// TwinCAT 3 PLC project BaseFBs
// Title: BaseFBs
// Company: Personal
// ProjectVersion: 1.0.0.3
// ProgramVersion: 3.1.4026.14
// libraries:
//   Tc2_Standard, * (Beckhoff Automation GmbH)
//   Tc2_System, * (Beckhoff Automation GmbH)
// project tree:
//   FBs/ FB_Base.TcPOU, FB_EquipmentBase.TcPOU, FB_Alarm.TcPOU, FB_SupervisorBase.TcPOU, ITF_Base.TcIO, ITF_EquipmentBase.TcIO, ITF_SupervisorBase.TcIO, Param_SupervisorBase.TcGVL
//   FBs/Structure/ ST_BaseDefinition.TcDUT, ST_EquipmentAlarm.TcDUT, ST_EquipmentAlarmListDetails.TcDUT
//   / PlcTask.TcTTO
//   POUs/ MAIN.TcPOU
//   TestFBs/TestBase/ FB_TestBase.TcPOU
//   TestFBs/TestEquipmentBase/ E_TestEquipmentAlarmList.TcDUT, FB_TestEquipmentBase.TcPOU
// real-time tasks:
//   TASK PlcTask: cycle T#10ms, priority 20, ADS port 350

CONFIGURATION BaseFBs
    RESOURCE PLC ON TwinCAT3
        TASK PlcTask(INTERVAL := T#10ms, PRIORITY := 20);
        PROGRAM MAIN WITH PlcTask : MAIN;
    END_RESOURCE
END_CONFIGURATION

// ---- FBs/Structure/ST_BaseDefinition.TcDUT
TYPE ST_BaseDefinition :
STRUCT
	Name		: STRING(40);
	Station		: string(40);
END_STRUCT
END_TYPE

// ---- FBs/Structure/ST_EquipmentAlarm.TcDUT
TYPE ST_EquipmentAlarm :
STRUCT
	Active			: BOOL;
	Message			: T_MaxString;
	Severity		: TcEventSeverity;
END_STRUCT
END_TYPE

// ---- FBs/Structure/ST_EquipmentAlarmListDetails.TcDUT
TYPE ST_EquipmentAlarmListDetails :
STRUCT
	FirstAlarm		: POINTER TO ST_EquipmentAlarm;
	AlarmListSize	: DINT; 
END_STRUCT
END_TYPE

// ---- TestFBs/TestEquipmentBase/E_TestEquipmentAlarmList.TcDUT
{attribute 'qualified_only'}
{attribute 'strict'}
{attribute 'to_string'}
TYPE E_TestEquipmentAlarmList :
(
	VerboseAlarm,
	InfoAlarm,
	WarningAlarm,
	ErrorAlarm,
	CriticalAlarm
);
END_TYPE

// ---- FBs/Param_SupervisorBase.TcGVL
{attribute 'qualified_only'}
VAR_GLOBAL CONSTANT
	AlarmListSize	: DINT := 50;
END_VAR

// ---- FBs/ITF_Base.TcIO
INTERFACE ITF_Base

PROPERTY Definition : REFERENCE TO ST_BaseDefinition
GET
END_GET
END_PROPERTY

PROPERTY EnableManualControl : Bool
SET
END_SET
END_PROPERTY

END_INTERFACE

// ---- FBs/ITF_EquipmentBase.TcIO
  INTERFACE ITF_EquipmentBase EXTENDS ITF_Base

PROPERTY AlarmListDetails : Reference to ST_EquipmentAlarmListDetails
GET
END_GET
END_PROPERTY

PROPERTY MainAlarm : Reference to ST_EquipmentAlarm
GET
END_GET
END_PROPERTY

METHOD Reset
END_METHOD

END_INTERFACE

// ---- FBs/ITF_SupervisorBase.TcIO
INTERFACE ITF_SupervisorBase

METHOD CheckAlarmCondition
VAR_INPUT
	AlarmToRaise		: ST_EquipmentAlarm;
	ConcatenateMessage	: T_MaxString;
END_VAR
END_METHOD

METHOD CheckAlarmConditionCustom
VAR_INPUT
	Active	: BOOL;
	Message	: T_MaxString;
	Severity	: TcEventSeverity;
END_VAR
END_METHOD

METHOD CompileAlarmList
VAR_INPUT
	AlarmListDetails		: ST_EquipmentAlarmListDetails;
END_VAR
END_METHOD

END_INTERFACE

// ---- POUs/MAIN.TcPOU
PROGRAM MAIN
VAR
	fbTestBase : FB_TestBase;
	fbTestEquipmentBase	: FB_TestEquipmentBase;
	fbTestEquipmentBase2	: FB_TestEquipmentBase;
	
	AnotherTestAlarmList	: ARRAY[E_TestEquipmentAlarmList.VerboseAlarm..E_TestEquipmentAlarmList.CriticalAlarm] OF ST_EquipmentAlarm;
	
	Reset	: BOOL;
	
	fbSupervistorBase : FB_SupervisorBase;
	
END_VAR

VAR PERSISTENT
	TestManualControl	: ARRAY[1..3] OF BOOL;
	TestName			: ARRAY[1..3] OF STRING(40);
	TestStation			: ARRAY[1..3] OF STRING(40);	
	

END_VAR

fbTestBase.Definition.Name := TestName[1];
fbTestBase.Definition.Station := TestStation[1];
fbTestBase.EnableManualControl := TestManualControl[1];

fbTestBase();

fbTestEquipmentBase.Definition.Name := TestName[2];
fbTestEquipmentBase.Definition.Station := TestStation[2];
fbTestEquipmentBase.EnableManualControl := TestManualControl[2];

fbTestEquipmentBase();

fbTestEquipmentBase2.Definition.Name := TestName[3];
fbTestEquipmentBase2.Definition.Station := TestStation[3];
fbTestEquipmentBase2.EnableManualControl := TestManualControl[3];

fbTestEquipmentBase2();

IF Reset THEN
	fbTestEquipmentBase.Reset();	
	fbTestEquipmentBase2.Reset();
	Reset := FALSE;
END_IF

fbSupervistorBase();

fbSupervistorBase.CompileAlarmList(AlarmListDetails := fbTestEquipmentBase.AlarmListDetails);
fbSupervistorBase.CompileAlarmList(AlarmListDetails := fbTestEquipmentBase2.AlarmListDetails);

END_PROGRAM

// ---- TestFBs/TestBase/FB_TestBase.TcPOU
FUNCTION_BLOCK FB_TestBase EXTENDS FB_Base

VAR
END_VAR

END_FUNCTION_BLOCK

// ---- FBs/FB_Base.TcPOU
FUNCTION_BLOCK ABSTRACT FB_Base IMPLEMENTS ITF_Base
VAR
	_Definition				: ST_BaseDefinition;
	_EnableManualControl	: BOOL;
END_VAR

PROPERTY Definition : REFERENCE TO ST_BaseDefinition
GET
Definition REF= _Definition;
END_GET
END_PROPERTY

PROPERTY EnableManualControl : BOOL
SET
_EnableManualControl := EnableManualControl;
END_SET
END_PROPERTY

END_FUNCTION_BLOCK

// ---- TestFBs/TestEquipmentBase/FB_TestEquipmentBase.TcPOU
FUNCTION_BLOCK FB_TestEquipmentBase EXTENDS FB_EquipmentBase
VAR
	TestAlarmList	: ARRAY[E_TestEquipmentAlarmList.VerboseAlarm..E_TestEquipmentAlarmList.CriticalAlarm] OF ST_EquipmentAlarm;
	
	AlarmType		: E_TestEquipmentAlarmList;
	RaiseAlarmFlag	: BOOL;
END_VAR


SUPER^();
fbAlarm(AlarmList := TestAlarmList);

IF RaiseAlarmFlag THEN
	
	CASE AlarmType OF
		E_TestEquipmentAlarmList.VerboseAlarm:
			_RaiseAlarm(AlarmToRaise := TestAlarmList[E_TestEquipmentAlarmList.VerboseAlarm], ConcatenateMessage := '');
		
		E_TestEquipmentAlarmList.InfoAlarm:
			_RaiseAlarm(AlarmToRaise := TestAlarmList[E_TestEquipmentAlarmList.InfoAlarm], ConcatenateMessage := '');
		
		E_TestEquipmentAlarmList.WarningAlarm:
			_RaiseAlarm(AlarmToRaise := TestAlarmList[E_TestEquipmentAlarmList.WarningAlarm], ConcatenateMessage := '');
		
		E_TestEquipmentAlarmList.ErrorAlarm:
			_RaiseAlarm(AlarmToRaise := TestAlarmList[E_TestEquipmentAlarmList.ErrorAlarm], ConcatenateMessage := '');
		
		E_TestEquipmentAlarmList.CriticalAlarm:
			_RaiseAlarm(AlarmToRaise := TestAlarmList[E_TestEquipmentAlarmList.CriticalAlarm], ConcatenateMessage := '');
		
	END_CASE

	RaiseAlarmFlag := FALSE;
END_IF

{warning 'Add method implementation '}
METHOD PROTECTED _GenerateAlarmList
TestAlarmList[E_TestEquipmentAlarmList.VerboseAlarm].Message 		:= 'Verbose Alarm';
TestAlarmList[E_TestEquipmentAlarmList.VerboseAlarm].Severity 		:= TcEventSeverity.Verbose;

TestAlarmList[E_TestEquipmentAlarmList.InfoAlarm].Message 			:= 'Info Alarm';
TestAlarmList[E_TestEquipmentAlarmList.InfoAlarm].Severity 			:= TcEventSeverity.Info;

TestAlarmList[E_TestEquipmentAlarmList.WarningAlarm].Message 		:= 'Warning Alarm';
TestAlarmList[E_TestEquipmentAlarmList.WarningAlarm].Severity 		:= TcEventSeverity.Warning;

TestAlarmList[E_TestEquipmentAlarmList.ErrorAlarm].Message 			:= 'Error Alarm';
TestAlarmList[E_TestEquipmentAlarmList.ErrorAlarm].Severity 		:= TcEventSeverity.Error;

TestAlarmList[E_TestEquipmentAlarmList.CriticalAlarm].Message 		:= 'Critical Alarm';
TestAlarmList[E_TestEquipmentAlarmList.CriticalAlarm].Severity 		:= TcEventSeverity.Critical;
END_METHOD

END_FUNCTION_BLOCK

// ---- FBs/FB_EquipmentBase.TcPOU
FUNCTION_BLOCK ABSTRACT FB_EquipmentBase EXTENDS FB_Base IMPLEMENTS ITF_EquipmentBase

VAR
	fbAlarm		: FB_Alarm;
	_MainAlarm	: ST_EquipmentAlarm;
	_AlarmListDetails	: ST_EquipmentAlarmListDetails;
	AlarmListUpperBound		: DINT;
	AlarmListLowerBound		: DINT;
	EmptyAlarmList			: BOOL;
	
	EquipmentBaseFirstScan	: BOOL := TRUE;
	
END_VAR

fbAlarm.Definition.Name := _Definition.Name;

_AlarmListDetails := fbAlarm.AlarmListDetails;

IF EquipmentBaseFirstScan THEN
	_GenerateAlarmList();
END_IF

EquipmentBaseFirstScan := FALSE;

METHOD PROTECTED _GenerateAlarmList
END_METHOD

METHOD PROTECTED _RaiseAlarm
VAR_INPUT
	AlarmToRaise	: REFERENCE TO ST_EquipmentAlarm;
	ConcatenateMessage	: T_MaxString;
END_VAR
AlarmToRaise.Active := TRUE;

IF (NOT _MainAlarm.Active) OR (AlarmToRaise.Severity > _MainAlarm.Severity) THEN
	_MainAlarm := AlarmToRaise;
	
	IF ConcatenateMessage <> '' THEN
		_MainAlarm.Message := CONCAT(STR1 := _MainAlarm.Message, STR2 := ConcatenateMessage);
	END_IF
	
END_IF
END_METHOD

{warning 'Add property implementation'}
PROPERTY AlarmListDetails : REFERENCE TO ST_EquipmentAlarmListDetails
GET
 AlarmListDetails REF= _AlarmListDetails;
END_GET
END_PROPERTY

{warning 'Add property implementation'}
PROPERTY MainAlarm : REFERENCE TO ST_EquipmentAlarm
GET
MainAlarm REF= _MainAlarm;
END_GET
END_PROPERTY

{warning 'Add method implementation '}
METHOD Reset
VAR
	ErrorIndex	: DINT;
END_VAR
_MainAlarm.Active := FALSE;
_MainAlarm.Severity := TcEventSeverity.Verbose;
_MainAlarm.Message := '';

fbAlarm.Reset();
END_METHOD

END_FUNCTION_BLOCK

// ---- FBs/FB_Alarm.TcPOU
FUNCTION_BLOCK  FB_Alarm EXTENDS FB_Base IMPLEMENTS ITF_Base
VAR_IN_OUT
	AlarmList	: ARRAY[*] OF ST_EquipmentAlarm;
END_VAR
VAR
	_AlarmListDetails	: ST_EquipmentAlarmListDetails;
	AlarmListUpperBound		: DINT;
	AlarmListLowerBound		: DINT;
	EmptyAlarmList			: BOOL;
	
	AlarmIndex				: DINT;
	DefinitionNameScanned	: BOOL := FALSE;
	
	FirstScan	: BOOL := TRUE;
END_VAR

_AlarmListHandling();

IF _Definition.Name <> '' AND not DefinitionNameScanned THEN
	
	FOR AlarmIndex := AlarmListLowerBound TO AlarmListUpperBound BY 1 DO
		AlarmList[AlarmIndex].Message := CONCAT(STR1 := ': ', STR2 := AlarmList[AlarmIndex].Message);
		AlarmList[AlarmIndex].Message := CONCAT(STR1 := _Definition.Name, STR2 := AlarmList[AlarmIndex].Message);
	END_FOR
	
	DefinitionNameScanned := TRUE;
END_IF

FirstScan := FALSE;

METHOD Private _AlarmListHandling

EmptyAlarmList := FALSE;
IF (SIZEOF(AlarmList) = 0) OR (AlarmList = 0) THEN
	EmptyAlarmList := TRUE;
	RETURN;
END_IF
	
IF FirstScan THEN	
	AlarmListLowerBound := LOWER_BOUND(AlarmList,1);
	AlarmListUpperBound := UPPER_BOUND(AlarmList,1);
	
	_AlarmListDetails.AlarmListSize := AlarmListUpperBound - AlarmListLowerBound + 1;
	_AlarmListDetails.FirstAlarm := ADR(AlarmList[AlarmListLowerBound]);
	
END_IF
END_METHOD

{warning 'Add property implementation'}
PROPERTY AlarmListDetails : REFERENCE TO ST_EquipmentAlarmListDetails
GET
 AlarmListDetails REF= _AlarmListDetails;
END_GET
END_PROPERTY

{warning 'Add method implementation '}
METHOD Reset
VAR
	ErrorIndex	: DINT;
END_VAR
IF EmptyAlarmList THEN
	RETURN;
END_IF

FOR ErrorIndex := AlarmListLowerBound TO AlarmListUpperBound BY 1 DO
	AlarmList[ErrorIndex].Active := FALSE;
END_FOR
END_METHOD

END_FUNCTION_BLOCK

// ---- FBs/FB_SupervisorBase.TcPOU
FUNCTION_BLOCK FB_SupervisorBase EXTENDS FB_EquipmentBase IMPLEMENTS ITF_SupervisorBase
VAR
	CompiledAlarm, CompiledAlarm_Intermediate		: ARRAY[0..Param_SupervisorBase.AlarmListSize] OF ST_EquipmentAlarm;	
	EmptyAlarm						: ST_EquipmentAlarm;	
	AlarmListIndex					: DINT;
	index							: DINT;
END_VAR

SUPER^();

_ResetAlarmList();

METHOD PRIVATE _ResetAlarmList
VAR_INPUT
END_VAR
MEMMOVE(destAddr := ADR(CompiledAlarm), srcAddr := ADR(CompiledAlarm_Intermediate), n := SIZEOF(CompiledAlarm));
MEMSET(destAddr := ADR(CompiledAlarm_Intermediate), fillByte := 0, n := SIZEOF(CompiledAlarm_Intermediate));
AlarmListIndex := 0;
END_METHOD

{warning 'Add method implementation '}
METHOD CheckAlarmCondition
VAR_INPUT
	AlarmToRaise		: ST_EquipmentAlarm;
	ConcatenateMessage	: T_MaxString;
END_VAR
SUPER^._RaiseAlarm(	AlarmToRaise := AlarmToRaise,
					ConcatenateMessage := ConcatenateMessage);
END_METHOD

{warning 'Add method implementation '}
METHOD CheckAlarmConditionCustom
VAR_INPUT
	Active	: BOOL;
	Message	: T_MaxString;
	Severity	: TcEventSeverity;
END_VAR
IF NOT Active THEN
	RETURN;
END_IF

_MainAlarm.Active := TRUE;

IF (Severity > _MainAlarm.Severity) THEN
	
	_MainAlarm.Severity := Severity;
	_MainAlarm.Message := Message;
	
END_IF
END_METHOD

{warning 'Add method implementation '}
METHOD CompileAlarmList
VAR_INPUT
	AlarmListDetails	: ST_EquipmentAlarmListDetails;
END_VAR

VAR
	MemoryPosition		: POINTER TO ST_EquipmentAlarm;
	i : DINT;

END_VAR
IF AlarmListIndex > Param_SupervisorBase.AlarmListSize THEN
	RETURN;
END_IF

IF AlarmListDetails.AlarmListSize = 0 THEN
	RETURN;
END_IF

IF AlarmListDetails.FirstAlarm = 0 THEN
	RETURN;
END_IF

FOR i := 0 TO (AlarmListDetails.AlarmListSize - 1) BY 1 DO
	
	MemoryPosition := AlarmListDetails.FirstAlarm + SIZEOF(EmptyAlarm)*i;
	
	IF MemoryPosition^.Active THEN
		CompiledAlarm_Intermediate[AlarmListIndex] := MemoryPosition^;
		AlarmListIndex := AlarmListIndex +1;
	END_IF

END_FOR
END_METHOD

END_FUNCTION_BLOCK
